TYPE T_Query_Interface : __SYSTEM.IQueryInterface; END_TYPE

(* stored: Version 1.1.0.1, ProductVersion 3.1.4024.4
   DUT T_Query_Interface: Id {70a001d6-4058-4f69-9b73-6b4158391c3c} *)
